TYPE "PLCtoMES_OP_ProcessData_OP220"
VERSION : 0.1
   STRUCT
      DATA : Real;
   END_STRUCT;

END_TYPE

